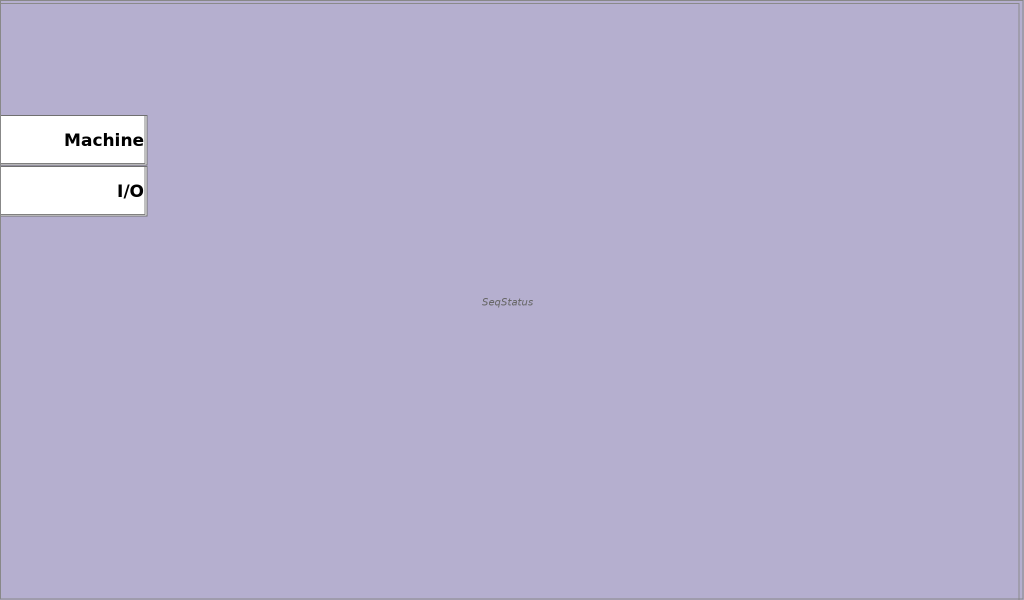
VISUALIZATION PLC_Status  // 1024x600
    Frame (-4,3 1023x598)
        shows SeqStatus()
        shows IO_Status()
        shows Test_Shuttle()
        shows Test_Place1()
        shows Test_Place2()
        shows Test_Place3()
        shows Test_Place4()
    Button (-3,115 150x50), "Machine", image: VisuSymbols.Symbols.Database2
        OnMouseDown: FrameSelectionChange Selection=SelectedFrame=eb142f5b-097c-4dbf-af2f-09085337604c, GlobSel=AssignDir=MainPage.GenElemInst_1003, AssignType=Directly, SelType=Locally
    Button (-3,166 150x50), "I/O", image: VisuSymbols.Symbols.Database2
        OnMouseDown: FrameSelectionChange Selection=SelectedFrame=eb142f5b-097c-4dbf-af2f-09085337604c, Selection=1, GlobSel=AssignDir=MainPage.GenElemInst_1003, AssignType=Directly, SelType=Locally
END_VISUALIZATION

(* stored: Version 1.1.0.1, ProductVersion 3.1.4024.12
   Visu PLC_Status: Id {4bd60ca1-a55e-45ec-a9dc-67b0f4099e23} *)
